TYPE UTime_t :
UNION
	dwValue  : ARRAY[0..1] OF DWORD;
	u64Value : ULINT;
END_UNION
END_TYPE

(* stored: Version 1.1.0.1, ProductVersion 3.1.4024.12
   DUT UTime_t: Id {49383c43-dc40-40bc-86d6-7fe4e4417591} *)
